# EPICS alarm handler configuration: alh_files/demo.alhConfig
GROUP NULL DEMO
$ALIAS Demo

GROUP DEMO GROUP1
CHANNEL  GROUP1  DEMO:PV1   -----
CHANNEL  GROUP1  DEMO:PV2   -----
CHANNEL  GROUP1  DEMO:PV3   -----

GROUP DEMO GROUP2
CHANNEL  GROUP2  DEMO:PV6   -----
CHANNEL  GROUP2  DEMO:PV7   -----

GROUP  GROUP2   GROUP3
CHANNEL  GROUP3  DEMO:PV4   -----
CHANNEL  GROUP3  DEMO:PV5   -----
